FUNCTION_BLOCK fbFCV
VAR_INPUT
	Interlock_1 : BOOL;
	Interlock_2 : BOOL;
	Interlock_3 : BOOL;
	Interlock_4 : BOOL;
	Interlock_5 : BOOL;
	Interlock_6 : BOOL;
	Interlock_7 : BOOL;

	AutoSp : REAL;
	ActPosIn : REAL;
END_VAR
VAR_OUTPUT
	ActPos : REAL;
	AutoMan : BOOL;
	FB_Open : BOOL;
	FB_Travelling : BOOL;
	FB_Close : BOOL;
	Alarm : BOOL;
	Alarm_ID : INT;

	CmdSpOut : REAL;
END_VAR
VAR
	Interlock_OK : BOOL;
	AutoReq : BOOL;
	ManReq : BOOL;
	ManSP : REAL;
	ManOpenReq : BOOL;
	ManCloseReq : BOOL;
	ManCmd : BOOL;
	rLowLimit : REAL;
	rLowLimitTol : REAL := 2;
	rHighLimit : REAL;
	rHighLimitTol : REAL := 2;

	strInterlock_1 : STRING;
	strInterlock_2 : STRING;
	strInterlock_3 : STRING;
	strInterlock_4 : STRING;
	strInterlock_5 : STRING;
	strInterlock_6 : STRING;
	strInterlock_7 : STRING;
	strAutoMan : STRING;
	strOpenTravClose : STRING;
	idxOpenTravClose : INT;
	EnableAlarm : BOOL;
	AlarmDelayTime : TIME := T#5S;
	tonAlarmDelay : TON;

	SimFCV : fbSimFCV;
END_VAR
VAR // added by the converter: edge detectors and wires of the graphical bodies
    _w1, _w2, _w3, _w4, _w5, _w6 : BOOL;
END_VAR

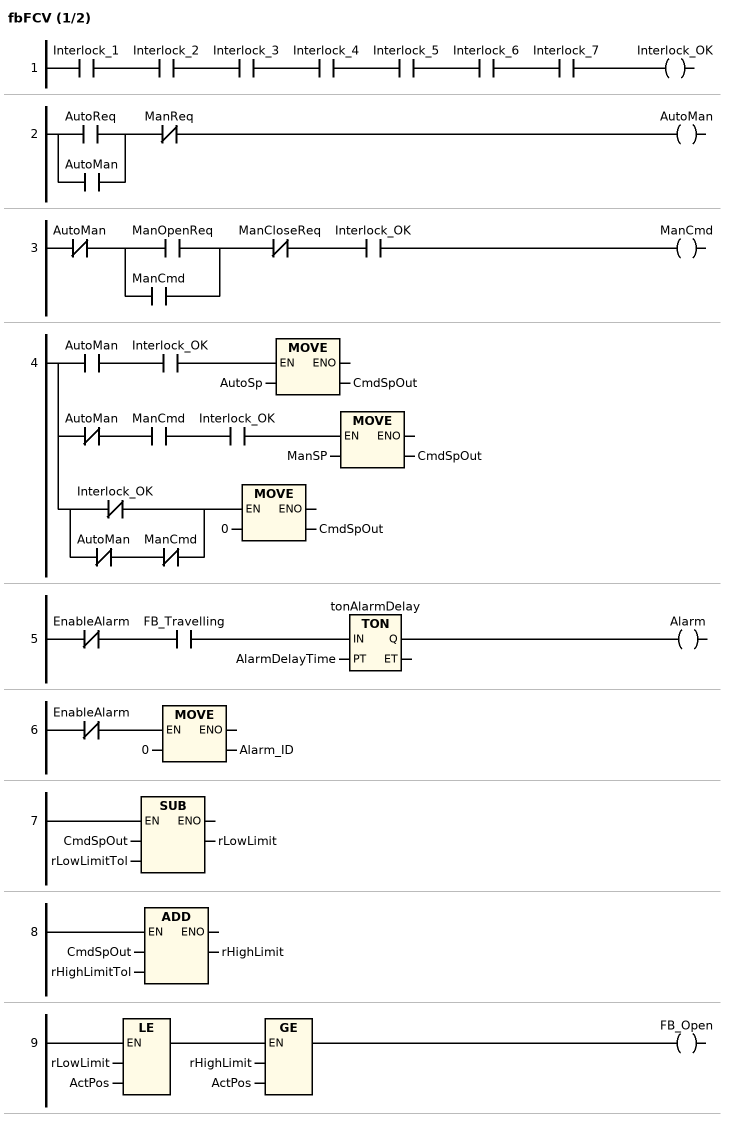
// NETWORK 1
Interlock_OK := Interlock_1 AND Interlock_2 AND Interlock_3 AND Interlock_4 AND Interlock_5 AND Interlock_6 AND Interlock_7;

// NETWORK 2
AutoMan := (AutoReq OR AutoMan) AND NOT ManReq;

// NETWORK 3
ManCmd := NOT AutoMan AND (ManOpenReq OR ManCmd) AND NOT ManCloseReq AND Interlock_OK;

// NETWORK 4
_w1 := AutoMan AND Interlock_OK;
IF _w1 THEN CmdSpOut := AutoSp; END_IF
_w2 := NOT AutoMan AND ManCmd AND Interlock_OK;
IF _w2 THEN CmdSpOut := ManSP; END_IF
_w3 := NOT Interlock_OK OR NOT AutoMan AND NOT ManCmd;
IF _w3 THEN CmdSpOut := 0; END_IF
(* _w1 OR _w2 OR _w3; result not used *)

// NETWORK 5
tonAlarmDelay(IN := NOT EnableAlarm AND FB_Travelling, PT := AlarmDelayTime); // TON
Alarm := tonAlarmDelay.Q;

// NETWORK 6
IF NOT EnableAlarm THEN Alarm_ID := 0; END_IF

// NETWORK 7
rLowLimit := CmdSpOut - rLowLimitTol;

// NETWORK 8
rHighLimit := CmdSpOut + rHighLimitTol;

// NETWORK 9
FB_Open := rLowLimit <= ActPos AND rHighLimit >= ActPos;

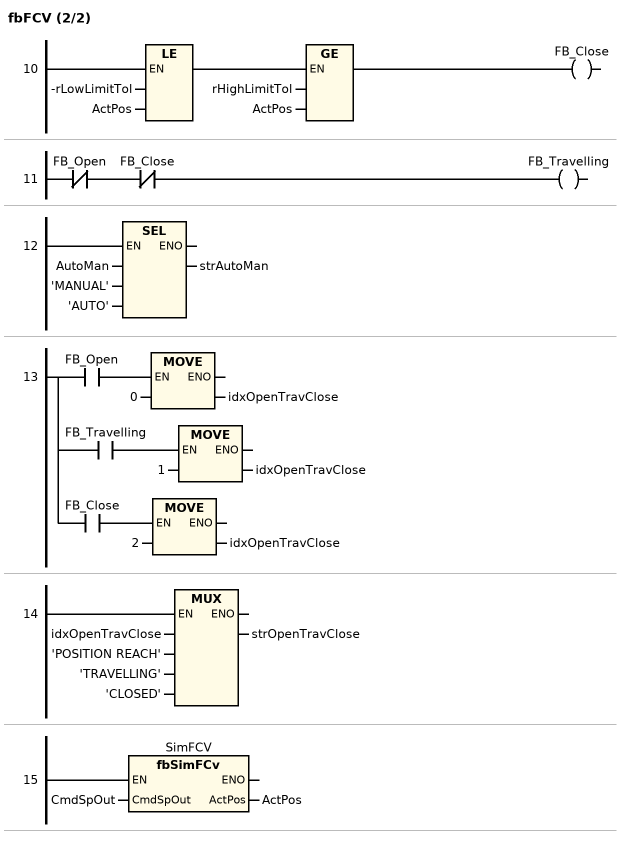
// NETWORK 10
FB_Close := (-rLowLimitTol) <= ActPos AND rHighLimitTol >= ActPos;

// NETWORK 11
FB_Travelling := NOT FB_Open AND NOT FB_Close;

// NETWORK 12
strAutoMan := SEL(AutoMan, 'MANUAL', 'AUTO');

// NETWORK 13
_w4 := FB_Open;
IF _w4 THEN idxOpenTravClose := 0; END_IF
_w5 := FB_Travelling;
IF _w5 THEN idxOpenTravClose := 1; END_IF
_w6 := FB_Close;
IF _w6 THEN idxOpenTravClose := 2; END_IF
(* _w4 OR _w5 OR _w6; result not used *)

// NETWORK 14
strOpenTravClose := MUX(idxOpenTravClose, 'POSITION REACH', 'TRAVELLING', 'CLOSED');

// NETWORK 15
SimFCV(CmdSpOut := CmdSpOut, ActPos => ActPos); // fbSimFCv

END_FUNCTION_BLOCK

(* stored: Version 1.1.0.1, ProductVersion 3.1.4022.17
   POU fbFCV: Id {a1ca00c2-4bc5-4464-b6b7-705d0549e8e4}, SpecialFunc None *)
